Universal Robots URScript: zaboj_fiala_program.script

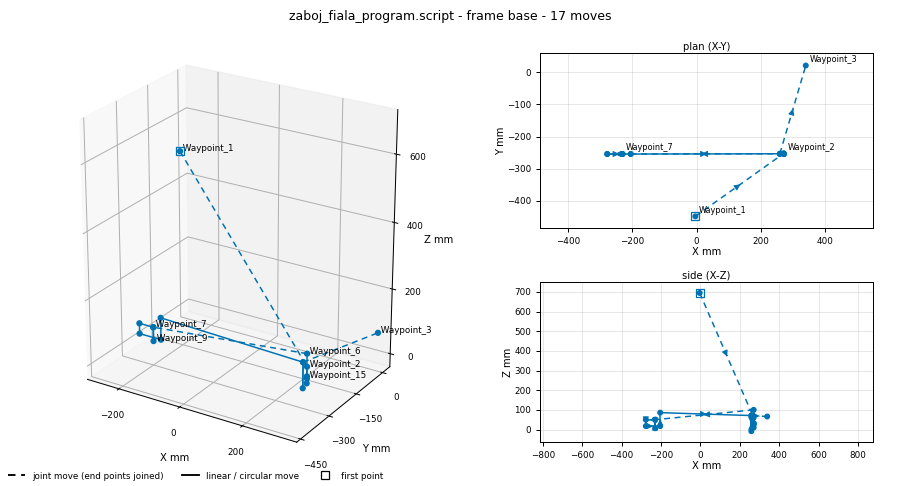
[picture p0: tool path of zaboj_fiala_program.script in frame base, 17 of 20 moves have a stored position in this frame; points joined in program order, loops and branches not executed]
def zaboj_fiala_program():
  global _hidden_verificationVariable=0
  step_count_39f631be_2866_4c45_90c6_6113dbd8747e = 0.0
  thread Step_Counter_Thread_8a2e1a7b_c817_435e_a248_d1a63734bcad():
    while (True):
      step_count_39f631be_2866_4c45_90c6_6113dbd8747e = step_count_39f631be_2866_4c45_90c6_6113dbd8747e + 1.0
      sync()
    end
  end
  run Step_Counter_Thread_8a2e1a7b_c817_435e_a248_d1a63734bcad()
  set_target_payload(1.110000, [0.000000, 0.000000, 0.054000], [0.001832, 0.001832, 0.001832, 0.000000, 0.000000, 0.000000])
  set_gravity([0.0, 0.0, 9.82])
  set_standard_analog_input_domain(0, 1)
  set_standard_analog_input_domain(1, 1)
  set_tool_analog_input_domain(0, 1)
  set_tool_analog_input_domain(1, 1)
  set_analog_outputdomain(0, 1)
  set_analog_outputdomain(1, 1)
  set_input_actions_to_default()
  set_tcp(p[3.414983750301692E-4,-7.378046129560278E-4,0.2251682051354249,-4.265841666109978E-5,-8.612665027929194E-6,-0.002773258026401147])
  set_tool_communication(True, 115200, 0, 1, 1.5, 3.5)
  set_tool_output_mode(0)
  set_tool_digital_output_mode(0, 1)
  set_tool_digital_output_mode(1, 1)
  set_tool_voltage(24)
  set_safety_mode_transition_hardness(1)
  global pocitadlo=7
  global var_2=0
  global referencePoint=p[0.27281535341285135,-0.001324543859192466,-0.05217449401005958,0.008705000024492312,-3.1415499774920335,4.921908573912826E-5]
  global separatorPoint=p[0.0,0.0,0.0,0.0,0.0,0.0]
  # begin: URCap Installation Node
  #   Source: UR Connect, 1.13.79, Universal Robots
  #   Type: UR Connect
  myurRPC = rpc_factory("xmlrpc","http://127.0.0.1:40474")
  # end: URCap Installation Node
  # begin: URCap Installation Node
  #   Source: Robotiq_Grippers, 3.19.1.111718, Robotiq Inc.
  #   Type: Vacuum
  #################################################
  # Vacuum Grip Check
  #################################################

  vacuumGripCheckThread1 = 0
  vacuumGripCheckThread2 = 0
  vacuumGripCheckThread3 = 0
  vacuumGripCheckThread4 = 0
  vacuumGripCheckThread1Running = False
  vacuumGripCheckThread2Running = False
  vacuumGripCheckThread3Running = False
  vacuumGripCheckThread4Running = False
  vacuumGripCheckslave_id = 1
  vacuumGripCheckThreadStarted = False

  thread vacuumGripCheck():
    slave_id = vacuumGripCheckslave_id
    vacuumGripCheckThreadStarted = True

    while (True):
      objectDetectedDebounceCtr = 0

      while (objectDetectedDebounceCtr < 3):
        if(rq_is_vacuum_obj_detected_by_slave_id(slave_id=9)):
          objectDetectedDebounceCtr = objectDetectedDebounceCtr + 1
        else:
          objectDetectedDebounceCtr = 0
        end
        sleep(0.1)
      end

      objectNotDetectedDebounceCtr = 0

      while objectNotDetectedDebounceCtr < 3:
        if (not rq_is_vacuum_obj_detected_by_slave_id(slave_id=9)):
          objectNotDetectedDebounceCtr = objectNotDetectedDebounceCtr + 1
        else:
          objectNotDetectedDebounceCtr = 0
        end
        sleep(0.1)
      end

      socket_open("127.0.0.1",29999,"dashboardServerSocket")
      socket_send_line("pause","dashboardServerSocket")
      socket_send_string("popup Vacuum grip check has detected an object drop.", "dashboardServerSocket")
      socket_send_byte(10, "dashboardServerSocket")
      socket_close("dashboardServerSocket")

      sleep(0.008)
    end
  end

  def startVacuumGripCheckThread(slave_id=9):
    vacuumGripCheckslave_id = slave_id
    threadHandle = run vacuumGripCheck()
    waitForVacuumGripCheckThreadStarted()
    return threadHandle
  end

  def stopVacuumGripCheckThread(threadHandle):
    kill threadHandle
  end

  def waitForVacuumGripCheckThreadStarted():
    while (not(vacuumGripCheckThreadStarted)):
      sleep(0.008)
    end
    vacuumGripCheckThreadStarted = False
  end
  #################################################
  # End - Vacuum Grip Check
  #################################################

  #################################################
  # Stops the pump on a distance travelled
  #################################################
  global stopPumpDistance = 100
  global stopPumpslave_id = 0
  global stopPumpThreadStarted = [False, False, False, False]
  global stopPumpThreadHandles = [0, 0, 0, 0]

  thread stopPumpOnDistanceTravelled():
    distance = stopPumpDistance
    slave_id = stopPumpslave_id
    stopPumpThreadStarted[rq_slave_id_to_index(slave_id)] = True

    measuredDistance = waitForDistanceTravelled(distance)

    rq_stop(slave_id_to_gripper_socket(slave_id))

    stopPumpThreadStarted[rq_slave_id_to_index(slave_id)] = False
  end

  def waitForDistanceTravelled(distance):
    startingPose = get_actual_tcp_pose()
    measuredDistance = 0
    while (measuredDistance < distance):
      sleep(0.1)
      measuredDistance = point_dist(get_actual_tcp_pose(), startingPose)
    end

    return measuredDistance
  end

  def startStopPumpOnDistanceTravelledThread(distance, slave_id=9):
    if (stopPumpThreadStarted[rq_slave_id_to_index(slave_id)]):
      return 0
    end

    global stopPumpDistance = distance
    global stopPumpslave_id = slave_id
    stopPumpThreadHandles[rq_slave_id_to_index(slave_id)] = run stopPumpOnDistanceTravelled()
    waitForStopPumpOnDistanceTravelledThreadStarted(slave_id)
    return stopPumpThreadHandles[rq_slave_id_to_index(slave_id)]
  end

  def waitForStopPumpOnDistanceTravelledThreadStarted(slave_id=9):
    while (not(stopPumpThreadStarted[rq_slave_id_to_index(slave_id)])):
      sleep(0.008)
    end
  end

  def stopStopPumpOnDistanceTravelledThread(slave_id=9):
    handle = stopPumpThreadHandles[rq_slave_id_to_index(slave_id)]
    threadIsRunning = stopPumpThreadStarted[rq_slave_id_to_index(slave_id)]
    if (threadIsRunning):
      kill handle
      stopPumpThreadHandles[rq_slave_id_to_index(slave_id)] = 0
    end
  end
  #################################################
  # End - Stops the pump on a distance travelled
  #################################################

  #################################################
  # Vacuum general functions
  #################################################
  def rq_wait_for_vacuum_object_detected(slave_id=9):
      while (not rq_is_vacuum_obj_detected_by_slave_id(slave_id)):
          if (rq_is_vacuum_timeout(slave_id)):
              return False
          end
          sleep(0.008)
      end
      return True
  end

  def rq_wait_for_vacuum_object_secured(slave_id=9):
      while (not rq_is_vacuum_obj_secured(slave_id)):
          if (rq_is_vacuum_timeout(slave_id)):
              return False
          end
          sleep(0.008)
      end
      return True
  end

  def rq_wait_for_vacuum_object_suction_complete(slave_id=9):
      remaining_retries = 50

       # Wait for suction started
      while (not rq_is_vacuum_obj_in_suction(slave_id) and
             not rq_is_vacuum_obj_detected_by_slave_id(slave_id) and
             remaining_retries > 0):
          sleep(0.01)
          remaining_retries = remaining_retries - 1
      end

      # Wait for suction completed
      while (rq_is_vacuum_obj_in_suction(slave_id)):
          if (rq_is_vacuum_timeout(slave_id)):
              return False
          end
          sleep(0.01)
      end

      return True
  end

  def rq_wait_for_vacuum_object_not_detected(slave_id=9):
      while (rq_is_vacuum_obj_detected_by_slave_id(slave_id)):
          sleep(0.01)
      end
  end

  def rq_is_vacuum_obj_detected_by_slave_id(slave_id=9):
      gOBJ = driver_gripper_client.getObjectDetectionFlag(slave_id)
      return is_vacuum_OBJ_object_detected(gOBJ)
  end

  def rq_is_vacuum_obj_detected(gripper_socket="1"):
      slave_id = gripper_socket_to_slave_id(gripper_socket)
      return rq_is_vacuum_obj_detected_by_slave_id(slave_id)
  end

  def rq_is_vacuum_obj_secured(slave_id=9):
      gOBJ = driver_gripper_client.getObjectDetectionFlag(slave_id)
      return is_vacuum_OBJ_object_secured(gOBJ)
  end

  def rq_is_vacuum_obj_in_suction(slave_id=9):
      gOBJ = driver_gripper_client.getObjectDetectionFlag(slave_id)
      return is_vacuum_OBJ_object_in_motion(gOBJ)
  end

  def rq_is_vacuum_timeout(slave_id=9):
      gFLT = driver_gripper_client.getFault(slave_id)
      return gFLT == 6
  end

  def is_vacuum_OBJ_object_in_motion(gOBJ):
      return gOBJ == 0
  end

  def is_vacuum_OBJ_object_detected(gOBJ):
      return gOBJ == 1 or gOBJ == 2
  end

  def is_vacuum_OBJ_object_secured(gOBJ):
      return gOBJ == 2
  end

  def rq_set_vacuum_and_wait(pressure, timeout, minimum, advanced_mode, slave_id=9):
      driver_gripper_client.configureVacuum(slave_id, advanced_mode, pressure, minimum, timeout)
  end

  def is_continuous_grip(maximum_vacuum):
    return maximum_vacuum == 0
  end

  def rq_vacuum_release(advanced_mode=False, shutoff_distance_cm=5, wait_for_object_released=True, gripper_socket="1"):
    rq_wait_for_gripper_reconnection()
    local slave_id = gripper_socket_to_slave_id(gripper_socket)
    local shutoff_distance = scale(shutoff_distance_cm, [0, 99], [0.00, 0.99])
    local pressure = 255
    local minimum = 0
    local timeout = 255
    rq_vacuum_release_raw(advanced_mode, pressure, minimum, timeout, shutoff_distance, wait_for_object_released, slave_id)
  end

  def rq_vacuum_release_raw(advanced_mode, pressure, minimum, timeout, shutoff_distance, wait_for_object_released, slave_id):
    rq_reset_fault_and_activate(slave_id)

    if advanced_mode:
      rq_set_vacuum_and_wait(pressure, timeout, minimum, 1, slave_id)
    else:
      rq_set_vacuum_and_wait(pressure, timeout, minimum, 0, slave_id)
    end

    # The following patch is for Robotiq's Camera issue when communication is lost, but not the activation
    # the communication driver reset the GTO bit
    driver_gripper_client.goto(slave_id, 1)

    if wait_for_object_released:
      while (rq_is_vacuum_obj_detected_by_slave_id(slave_id)):

        if advanced_mode:
          rq_set_vacuum_and_wait(pressure, timeout, minimum, 1, slave_id)
        else:
          rq_set_vacuum_and_wait(pressure, timeout, minimum, 0, slave_id)
        end

        # The following patch is for Robotiq's Camera issue when communication is lost, but not the activation
        # the communication driver reset the GTO bit
        driver_gripper_client.goto(slave_id, 1)
        sleep(0.01)
      end
    end

    if advanced_mode:
      startStopPumpOnDistanceTravelledThread(shutoff_distance, slave_id)
    end
  end

  def rq_vacuum_grip(advanced_mode=False, maximum_vacuum=60, minimum_vacuum=40, timeout_ms=3000, wait_for_object_detected=True, gripper_socket="1"):
    rq_wait_for_gripper_reconnection()
    local slave_id = gripper_socket_to_slave_id(gripper_socket)
    local pressure = floor(scale(maximum_vacuum, [0, 100], [100, 0]))
    local minimum = floor(scale(minimum_vacuum, [0, 100], [100, 0]))
    local timeout = floor(scale(timeout_ms, [0, 25500], [0, 255]))
    rq_vacuum_grip_raw(advanced_mode, pressure, minimum, timeout, slave_id)
    if wait_for_object_detected:
          suction_completed = rq_wait_for_vacuum_object_suction_complete(slave_id)
          if(not suction_completed):
            driver_gripper_client.goto(slave_id, 0)
          end
    end
  end

  def rq_vacuum_grip_raw(advanced_mode, pressure, minimum, timeout, slave_id):
    stopStopPumpOnDistanceTravelledThread(slave_id)
    rq_reset_fault_and_activate(slave_id)

    if advanced_mode:
      rq_set_vacuum_and_wait(pressure, timeout, minimum, 1, slave_id)
    else:
      rq_set_vacuum_and_wait(pressure, timeout, minimum, 0, slave_id)
    end

    driver_gripper_client.goto(slave_id, 1)
  end

  def is_FLT_no_fault(gFLT):
      return gFLT == 0
  end

  def is_FLT_vacuum_timeout(gFLT):
    return gFLT == 6
  end

  def is_FLT_faulted(gFLT):
      return gFLT >= 8
  end

  def rq_reset_fault_and_activate(slave_id):
      gFLT = driver_gripper_client.getFault(slave_id)

      if(not is_FLT_no_fault(gFLT)):
          if(is_FLT_vacuum_timeout(gFLT)):
              driver_gripper_client.goto(slave_id, 0)
          elif(is_FLT_faulted(gFLT)):
              driver_gripper_client.goto(slave_id, 0)
              driver_gripper_client.activate([slave_id], True)
          end
      elif(not rq_is_gripper_activated(slave_id)):
          driver_gripper_client.goto(slave_id, 0)
          driver_gripper_client.activate([slave_id], False)
      end
  end
  #################################################
  # End - Vacuum general functions
  #################################################
    def scale(value, rawRange, scaledRange):
        def computeSlope(inputRange, outputRange):
            outputRangeDelta = outputRange[1] - outputRange[0]
            inputRangeDelta = inputRange[1] - inputRange[0]

            if (inputRangeDelta == 0):
                return 0
            else:
                return outputRangeDelta / inputRangeDelta
            end
        end

        def computeIntercept(slope, inputRange, outputRange):
            return outputRange[0] - (slope * inputRange[0])
        end

        def clipScaledValue(outputScaledValue, outputRange):
            if (outputRange[0] < outputRange[1]):
                return clipWhenLowerLimitIsLessThanHigher(outputScaledValue, outputRange)
            else:
                return clipWhenLowerLimitIsGreaterThanHigherLimit(outputScaledValue, outputRange)
            end
        end

        def clipWhenLowerLimitIsGreaterThanHigherLimit(outputScaledValue, outputRange):
            if (outputScaledValue < outputRange[1]):
                return outputRange[1]
            elif (outputScaledValue > outputRange[0]):
                return outputRange[0]
            else:
                return outputScaledValue
            end
        end

        def clipWhenLowerLimitIsLessThanHigher(outputScaledValue, outputRange):
            if (outputScaledValue < outputRange[0]):
                return outputRange[0]
            elif (outputScaledValue > outputRange[1]):
                return outputRange[1]
            else:
                return outputScaledValue
            end
        end

        slope = computeSlope(rawRange, scaledRange)
        intercept = computeIntercept(slope, rawRange, scaledRange)
        scaledValue = slope * value + intercept
        return clipScaledValue(scaledValue, scaledRange)
    end

    def limit(value, range):
        return scale(value, range, range)
    end

  vacuumGripCheckWarningTitle = "Vacuum grip check"
  vacuumGripCheckWarningMessage = "Vacuum gripper object lost"
  vacuumGripTimeoutTitle = "Vacuum gripper fault"
  vacuumGripTimeoutMessage = "Grip has timed out"
  # end: URCap Installation Node
  # begin: URCap Installation Node
  #   Source: Robotiq_Grippers, 3.19.1.111718, Robotiq Inc.
  #   Type: Gripper
  RQ_UNIT_PERCENT = 0
  RQ_UNIT_MM = 1
  RQ_UNIT_INCH = 2

  global gripper_reconnecting = False
  rq_current_limit_enabled = False
  gripper_closed_norm = [100, 100, 100, 100]
  gripper_open_norm = [0, 0, 0, 0]
  gripper_closed_mm = [0, 0, 0, 0]
  gripper_open_mm = [50, 50, 50, 50]

  driver_gripper_client = rpc_factory("xmlrpc","http://127.0.0.1:63353")

  def rq_set_force_norm(force_norm, gripper_socket="1"):
      rq_wait_for_gripper_reconnection()
      slave_id = gripper_socket_to_slave_id(gripper_socket)
      rq_set_force_norm_multi_grippers(force_norm, [slave_id])
  end

  def rq_set_force_norm_multi_grippers(force_norm, slave_ids=[9]):
      driver_gripper_client.setForce(slave_ids, force_norm)
  end

  def rq_set_speed_norm(speed_norm, gripper_socket="1"):
      rq_wait_for_gripper_reconnection()
      slave_id = gripper_socket_to_slave_id(gripper_socket)
      rq_set_speed_norm_multi_grippers(speed_norm, [slave_id])
  end

  def rq_set_speed_norm_multi_grippers(speed_norm, slave_ids=[9]):
      driver_gripper_client.setSpeed(slave_ids, speed_norm)
  end

  def rq_open_and_wait(gripper_socket="1"):
      rq_wait_for_gripper_reconnection()
      slave_id = gripper_socket_to_slave_id(gripper_socket)
      driver_gripper_client.openGripper(slave_id)
      rq_wait_for_motion_complete([slave_id])
  end

  def rq_close_and_wait(gripper_socket="1"):
      rq_wait_for_gripper_reconnection()
      slave_id = gripper_socket_to_slave_id(gripper_socket)
      driver_gripper_client.closeGripper(slave_id)
      rq_wait_for_motion_complete([slave_id])
  end

  def rq_move_norm_multi_grippers(position, slave_ids=[9]):
     # rq_wait_for_gripper_reconnection fucntion is not called here because it is already done in the gripper contribution
     # script and this function is not defined for public usage.
     all_gripper_limits = get_all_gripper_limits(slave_ids)
     driver_gripper_client.move(slave_ids, position, RQ_UNIT_PERCENT, all_gripper_limits)
  end

  def rq_move_and_wait_norm_multi_grippers(position, slave_ids=[9]):
       all_gripper_limits = get_all_gripper_limits(slave_ids)
       driver_gripper_client.move(slave_ids, position, RQ_UNIT_PERCENT, all_gripper_limits)
       rq_wait_for_motion_complete(slave_ids)
  end

  def rq_move_and_wait(position, unit, gripper_socket="1"):
     rq_wait_for_gripper_reconnection()
     slave_id = gripper_socket_to_slave_id(to_str(gripper_socket))
     all_gripper_limits = get_all_gripper_limits([slave_id])
     driver_gripper_client.move([slave_id], position, unit, all_gripper_limits)
     rq_wait_for_motion_complete([slave_id])
  end

  def rq_move_and_wait_norm(position, gripper_socket="1"):
      rq_move_and_wait(position, RQ_UNIT_PERCENT, gripper_socket)
  end

  def rq_move_and_wait_mm(position, gripper_socket="1"):
      rq_move_and_wait(position, RQ_UNIT_MM, gripper_socket)
  end

  def rq_move_and_wait_inches(position, gripper_socket="1"):
     rq_move_and_wait(position, RQ_UNIT_INCH, gripper_socket)
  end

  def rq_is_object_detected(gripper_socket="1"):
     slave_id = gripper_socket_to_slave_id(gripper_socket)
     return driver_gripper_client.isObjectDetected(slave_id)
  end

  def rq_current_pos_norm(gripper_socket="1"):
      slave_id = gripper_socket_to_slave_id(gripper_socket)
      gripper_limits = get_gripper_limits(gripper_socket)
      return driver_gripper_client.getCurrentPosition(slave_id,
                                    RQ_UNIT_PERCENT,
                                    gripper_limits[0],
                                    gripper_limits[1],
                                    gripper_limits[2],
                                    gripper_limits[3])
  end

  def rq_current_pos_mm(gripper_socket=1):
      slave_id = gripper_socket_to_slave_id(to_str(gripper_socket))
      gripper_limits = get_gripper_limits(to_str(gripper_socket))
      return driver_gripper_client.getCurrentPosition(slave_id,
                                    RQ_UNIT_MM,
                                    gripper_limits[0],
                                    gripper_limits[1],
                                    gripper_limits[2],
                                    gripper_limits[3])
  end

  def rq_current_pos_inches(gripper_socket=1):
      slave_id = gripper_socket_to_slave_id(to_str(gripper_socket))
      gripper_limits = get_gripper_limits(to_str(gripper_socket))
      return driver_gripper_client.getCurrentPosition(slave_id,
                                    RQ_UNIT_INCH,
                                    gripper_limits[0],
                                    gripper_limits[1],
                                    gripper_limits[2],
                                    gripper_limits[3])
  end

  def rq_reset(gripper_socket="1"):
      slave_id = gripper_socket_to_slave_id(gripper_socket)
      driver_gripper_client.deactivate([slave_id])
  end

  def rq_set_gripper_max_cur(current_mA, gripper_socket="1"):
      rq_wait_for_gripper_reconnection()
      slave_id = gripper_socket_to_slave_id(gripper_socket)
      driver_gripper_client.setMaximumCurrent(current_mA, slave_id)
  end

  def rq_get_gripper_max_cur(gripper_socket="1"):
      slave_id = gripper_socket_to_slave_id(gripper_socket)
      return driver_gripper_client.getMaximumCurrent(slave_id)
  end

  def rq_set_max_current_for_all_grippers():
      rq_wait_for_gripper_reconnection()
      driver_gripper_client.setMaximumCurrentOnAllGrippers(rq_current_limit_enabled)
  end

  def rq_is_gripper_activated(slave_id=9):
      return driver_gripper_client.isGripperActivated(slave_id)
  end

  def rq_is_gripper_connected(slave_id=9):
      return driver_gripper_client.isGripperConnected(slave_id)
  end

  def rq_get_fault(slave_id=9):
      return driver_gripper_client.getFault(slave_id)
  end

  def rq_activate_and_wait(gripper_socket="1"):
      slave_id = gripper_socket_to_slave_id(gripper_socket)
      if (not rq_is_gripper_activated(slave_id)):
        driver_gripper_client.activate([slave_id], False)
      end
  end

  def rq_activate_all_grippers(reset=False):
      empty_array_used_to_act_on_all_grippers = []
      if (reset):
        driver_gripper_client.activate(empty_array_used_to_act_on_all_grippers, True)
      else:
        driver_gripper_client.activateIfRequired(empty_array_used_to_act_on_all_grippers)
      end
  end

  def get_closed_norm(gripper_socket):
      return gripper_closed_norm[rq_gripper_socket_to_index(gripper_socket)]
  end

  def get_open_norm(gripper_socket):
      return gripper_open_norm[rq_gripper_socket_to_index(gripper_socket)]
  end

  def get_open_mm(gripper_socket):
      return gripper_open_mm[rq_gripper_socket_to_index(gripper_socket)]
  end

  def get_closed_mm(gripper_socket):
      return gripper_closed_mm[rq_gripper_socket_to_index(gripper_socket)]
  end

  def set_closed_norm(closed_norm, gripper_socket):
      gripper_closed_norm[rq_gripper_socket_to_index(gripper_socket)] = closed_norm
  end

  def set_open_norm(open_norm, gripper_socket):
      gripper_open_norm[rq_gripper_socket_to_index(gripper_socket)] = open_norm
  end

  def set_closed_mm(closed_mm, gripper_socket):
      gripper_closed_mm[rq_gripper_socket_to_index(gripper_socket)] = closed_mm
  end

  def set_open_mm(opened_mm, gripper_socket):
      gripper_open_mm[rq_gripper_socket_to_index(gripper_socket)] = opened_mm
  end

  def slave_id_to_gripper_socket(slave_id):
      if slave_id == 9:
          return "1"
      else:
          return to_str(slave_id)
      end
  end

  def gripper_socket_to_slave_id(gripper_socket):
      if gripper_socket == "1":
          return 9
      else:
          return to_num(gripper_socket)
      end
  end

  def rq_slave_id_to_index(slave_id):
      if slave_id == 9:
          return 0
      else:
          return slave_id - 1
      end
  end

  def rq_gripper_socket_to_index(gripper_socket):
      return to_num(gripper_socket) - 1
  end

  def get_all_gripper_limits(slave_ids):
     all_gripper_limits = [0, 0, 0, 0, 0, 0, 0, 0, 0, 0, 0, 0, 0, 0, 0, 0]
     nb_slave_ids = get_list_length(slave_ids)
     slave_id_index = 0
     index = 0
     sub_index = 0
     while (index < nb_slave_ids):
         slave_id_index = 0
         items_per_limit = 4
         gripper_socket = slave_id_to_gripper_socket(slave_ids[index])
         gripper_limits = get_gripper_limits(gripper_socket)
         while (sub_index < items_per_limit):
            all_gripper_limits[index] = gripper_limits[sub_index]
            sub_index = sub_index + 1
            index = index + 1
         end
         index = index + 1
     end

     return all_gripper_limits
  end

  def get_gripper_limits(gripper_socket):
      return [get_closed_norm(gripper_socket),
              get_open_norm(gripper_socket),
              get_closed_mm(gripper_socket),
              get_open_mm(gripper_socket)]
  end

  def rq_wait_for_motion_complete(slave_ids):
      nb_slave_ids = get_list_length(slave_ids)
      index = 0
      while (index < nb_slave_ids):
        rq_wait(slave_ids[index])
        index = index + 1
      end
  end

  def rq_stop(gripper_socket="1"):
      slave_id = gripper_socket_to_slave_id(gripper_socket)
      driver_gripper_client.goto(slave_id, 0)
  end

  def rq_wait(slave_id):
      # Wait for the gripper motion to complete
      while (not rq_is_motion_complete(slave_id)):
          # The following patch is for Robotiq's Camera issue when communication is lost, but not the activation
          # the communication driver reset the GTO bit
          driver_gripper_client.goto(slave_id, 1)
          sleep(0.1)
      end
  end

  def rq_is_motion_complete(slave_id):
      detection_flag = driver_gripper_client.getObjectDetectionFlag(slave_id)
      return detection_flag > 0 and detection_flag < 4
  end

  def write_error_popup(index, message_part_1, message_part_2, title):
      popup_message_part_1 = str_cat(message_part_1, index)
      popup_message_part_2 = str_cat(popup_message_part_1, " ")
      popup_message = str_cat(popup_message_part_2, message_part_2)
      return popup(popup_message, title, False, True, True)
  end

  def rq_disconnect_grippers():
      driver_gripper_client.pauseAndDisconnect()
  end

  def rq_reconnect_grippers(blocking=False, slave_ids=[]):
      if blocking:
          global gripper_reconnecting = True
          driver_gripper_client.reconnectAndResume(slave_ids)
          gripper_reconnecting = False
      else:
          thread recon_thread():
              rq_reconnect_grippers(True)
              return False
          end
          thrd = run recon_thread()
      end
  end

  def rq_wait_for_gripper_reconnection(timeout_s = 30.0):
      while (gripper_reconnecting == True):
          if (timeout_s <= 0):
            popup("Gripper has not reconnected before the expected time")
            halt
          else:
            sync()
            timeout_s = timeout_s - get_steptime()
          end
      end
  end

  def rq_gripper_allow_tool_com(allow_tool_comm):
      driver_gripper_client.allowToolComm(allow_tool_comm)
  end
  set_closed_norm(100.0, "1")
  set_open_norm(0.0, "1")
  set_closed_mm(0.0, "1")
  set_open_mm(50.0, "1")
  set_closed_norm(100.0, "2")
  set_open_norm(0.0, "2")
  set_closed_mm(0.0, "2")
  set_open_mm(50.0, "2")
  set_closed_norm(100.0, "3")
  set_open_norm(0.0, "3")
  set_closed_mm(0.0, "3")
  set_open_mm(50.0, "3")
  set_closed_norm(100.0, "4")
  set_open_norm(0.0, "4")
  set_closed_mm(0.0, "4")
  set_open_mm(50.0, "4")
  rq_current_limit_enabled = False
  # end: URCap Installation Node
  global Pallet_1_cnt=1
  global Pallet_1_lct=1
  global Pallet_1_lno=1
  global Pallet_1_sep= False
  global Pallet_1_tct=1
  global qNearApproach=[0,0,0,0,0,0]
  global Waypoint_1_p=p[-.003732499146, -.447764350544, .694668676500, .010357527271, 2.217455435209, -2.215428702531]
  global Waypoint_1_q=[0.004420539364218712, -1.5699242066223924, 0.010914627705709279, -1.5611537259868165, -0.009149853383199513, -0.008998696004049123]
  global Waypoint_2_p=p[.270561572388, -.252460408212, .060750519249, -2.205633529341, 2.237137668558, .000000000220]
  global Waypoint_2_q=[-0.38798117147393185, -1.7670171967297028, -1.4314454771594134, -1.5127431085216578, 1.5630238713731401, -0.37426215443183697]
  global Waypoint_15_p=p[.270561572385, -.252460408216, .025108204613, -2.205633532066, 2.237137671479, .000000000266]
  global Waypoint_15_q=[-0.387640232785321, -1.7878663927529868, -1.574689349085693, -1.3486454019375724, 1.5632032959842548, -0.37526689414023995]
  global Waypoint_4_p=p[.271723132448, -.254713739484, .032576839225, -2.202352738203, 2.233984750329, -.017109190704]
  global Waypoint_4_q=[-0.39231975839608957, -1.777546052304718, -1.5566950178122445, -1.365160337822867, 1.5630833526801635, -0.37973253437504706]
  global Waypoint_5_p=p[.270561572159, -.253261773950, .010467803518, -2.205633542175, 2.237137697756, .000000006507]
  global Waypoint_5_q=[-0.3896634195662285, -1.805539464463246, -1.6233792723820244, -1.2822808384995135, 1.5633685440948906, -0.377819460409726]
  global Waypoint_6_p=p[.270561572150, -.253261773946, .100610117048, -2.205633531713, 2.237137687145, .000000006506]
  global Waypoint_6_q=[-0.39059338186191184, -1.7752166803415488, -1.2341938193302262, -1.7018008441992443, 1.5631981308940244, -0.3753075181511152]
  global Waypoint_7_p=p[-.230058808373, -.254188582133, .050546411075, -2.205633551354, 2.237137688707, -.000000002111]
  global Waypoint_7_q=[-1.9158549360473138, -1.6556048584721488, -1.6085609835301513, -1.4470858589855453, 1.5627141197324992, -1.9027213849297713]
  global Waypoint_9_p=p[-.230058808390, -.254188582182, .007047120969, -2.205633540891, 2.237137678096, -.000000002113]
  global Waypoint_9_q=[-1.9154641598153326, -1.6964409636789144, -1.7725358360043462, -1.2422691400022003, 1.563132548677892, -1.9039956648963363]
  global Waypoint_11_p=p[-.277401121907, -.254188582125, .050546411070, -2.205633551354, 2.237137688707, -.000000002111]
  global Waypoint_11_q=[-2.045659040969955, -1.8025670740351707, -1.4352832270086573, -1.4734087088425873, 1.5631794833456076, -2.0322455626523688]
  global Waypoint_12_p=p[-.277401121893, -.254188582096, .018070817914, -2.205633540892, 2.237137678095, -.000000002109]
  global Waypoint_12_q=[-2.045358845597888, -1.825729367137832, -1.5604181602870781, -1.3251075677590576, 1.5633936278058413, -2.0331527047927835]
  global Waypoint_13_p=p[-.204474181310, -.254188582073, .018070817902, -2.205633551354, 2.237137688706, -.000000002109]
  global Waypoint_13_q=[-1.8362919914072373, -1.6095973638389953, -1.8134970852229308, -1.288148318123807, 1.5627547664611345, -1.8244687075886024]
  global Waypoint_14_p=p[-.204474181308, -.254188582064, .086413131433, -2.205633551354, 2.237137688706, -.000000002108]
  global Waypoint_14_q=[-1.8369625886427805, -1.574832125077247, -1.5248047019871604, -1.6116166051216325, 1.5624717189936659, -1.8224669010736845]
  global Waypoint_8_p=p[.258569396158, -.253443601432, .071606282054, -2.202406735368, 2.240314480847, -.000000000314]
  global Waypoint_8_q=[-0.4042975507105382, -1.7298519365980187, -1.4251167858707436, -1.5562383352509102, 1.5629115038954633, -0.38735228726952897]
  global Waypoint_10_p=p[.258569396172, -.253443601435, -.007836031423, -2.202406734996, 2.240314481213, -.000000000000]
  global Waypoint_10_q=[-0.4035716267056175, -1.7950209472926995, -1.7277873303001208, -1.1883889938254129, 1.5635490193420658, -0.3896017747848468]
  global Waypoint_3_p=p[.339173069408, .020646450111, .066698974081, -.046899901835, 3.140174557594, -.015225451020]
  global Waypoint_3_q=[0.46848809719085693, -1.6360541782774867, -1.5524871349334717, -1.5260256093791504, 1.5533761978149414, 2.0090246200561523]
  global Approach_p=p[.272815353377, -.001324543879, -.033905691191, .008705000027, -3.141549977485, .000049219079]
  global Approach_q=[0.5000229007972248, -1.457555270442966, -2.2252279375503816, -1.0285170994385489, 1.5629147840442803, 2.0609351731087564]
  global ToolActionPoint_p=p[.272815353413, -.001324543859, -.052174494010, .008705000022, -3.141549977485, .000049219087]
  global ToolActionPoint_q=[0.500250470542329, -1.5124229690085453, -2.280892902919593, -0.9179415944854314, 1.5635788131215058, 2.060298978026008]
  global Exit_1_p=p[.272815353404, -.001324543864, .045467820739, .008705000021, -3.141549977496, .000049219082]
  global Exit_1_q=[0.49925098394912215, -1.3352160082302609, -1.9246151993381408, -1.4514821535151832, 1.5615809977592896, 2.0636040213119218]
  $ 2 "BeforeStart"
  # begin: URCap Program Node
  #   Source: Robotiq_Grippers, 3.19.1.111718, Robotiq Inc.
  #   Type: Gripper Activate
  $ 3 "Gripper Reset and Activate"

  rq_set_max_current_for_all_grippers()

  reset_and_activate = True

  rq_activate_all_grippers(True)
  # end: URCap Program Node
  $ 4 "MoveJ"
  $ 5 "Waypoint_1" "breakAfter"
  movej(get_inverse_kin(Waypoint_1_p, qnear=Waypoint_1_q), a=1.3962634015954636, v=1.0471975511965976)
  $ 6 "Wait Sensor_vzadu=HI"
  while (get_standard_digital_in(2) == False):
    sync()
  end
  $ 66 "Thread_1"
  thread Thread_1():
    while (True):
      $ 67 "Set Dopravnik=On"
      set_standard_digital_out(2, True)
      $ 68 "Wait Sensor_vzadu=HI"
      while (get_standard_digital_in(2) == False):
        sync()
      end
      $ 69 "Set Dopravnik=Off"
      set_standard_digital_out(2, False)
      $ 70 "Wait Sensor_vzadu=LO"
      while (get_standard_digital_in(2) == True):
        sync()
      end
      $ 71 "Wait: 1.0"
      sleep(1.0)
    end
  end
  threadId_Thread_1 = run Thread_1()
  while (True):
    $ 7 "Robot Program"
    $ 8 "MoveJ"
    $ 9 "Waypoint_2" "breakAfter"
    movej(get_inverse_kin(Waypoint_2_p, qnear=Waypoint_2_q), a=1.3962634015954636, v=1.0471975511965976)
    $ 10 "Wait Sensor_vzadu=HI"
    while (get_standard_digital_in(2) == False):
      sync()
    end
    # begin: URCap Program Node
    #   Source: Robotiq_Grippers, 3.19.1.111718, Robotiq Inc.
    #   Type: Gripper
    $ 11 "Gripper Close (1)"
    gripper_slave_ids_0 = [9]
    popupErrorGripperWord = "Gripper"
    popupErrorNoConnection1 = "must be connected to run this program."
    popupErrorNoConnection2 = "No connection"
    popupErrorNotActivated1 = "is not activated. Go to Installation tab > Gripper to activate it and run the program again."
    popupErrorNotActivated2 = "Not activated"
    rq_gripper_speed = 100.0
    rq_gripper_force = 20.0
    rq_gripper_position = 100.0
    rq_is_blocking = True
    rq_is_robot_compliant = False
    nb_slave_ids = get_list_length(gripper_slave_ids_0)
    rq_wait_for_gripper_reconnection()
    index = 0
    while (index < nb_slave_ids):
        if (not rq_is_gripper_connected(gripper_slave_ids_0[index])):
            write_error_popup(index, popupErrorGripperWord, popupErrorNoConnection1, popupErrorNoConnection2)
        end
        index = index + 1
    end
    index = 0
    while (index < nb_slave_ids):
        if (not rq_is_gripper_activated(gripper_slave_ids_0[index])):
            write_error_popup(index, popupErrorGripperWord, popupErrorNotActivated1, popupErrorNotActivated2)
        end
        index = index + 1
    end
    rq_set_speed_norm_multi_grippers(rq_gripper_speed, gripper_slave_ids_0)
    rq_set_force_norm_multi_grippers(rq_gripper_force, gripper_slave_ids_0)
    if (rq_is_blocking):
        if rq_is_robot_compliant:
            zero_ftsensor()
            sleep(0.02)
            # Maximum allowed deviation values for non-compliant axes are default values generated by UR in a Force node
            force_mode(tool_pose(), [1, 1, 0, 0, 0, 0], [0.0, 0.0, 0.0, 0.0, 0.0, 0.0], 2, [0.15, 0.15, 0.1, 0.3490658503988659, 0.3490658503988659, 0.3490658503988659])
        end
        rq_move_and_wait_norm_multi_grippers(rq_gripper_position, gripper_slave_ids_0)
        if rq_is_robot_compliant:
            end_force_mode()
        end
    else:
        rq_move_norm_multi_grippers(rq_gripper_position, gripper_slave_ids_0)
    end
    # end: URCap Program Node
    $ 12 "MoveL"
    $ 13 "Waypoint_15" "breakAfter"
    movel(Waypoint_15_p, a=1.2, v=0.05)
    $ 14 "var_1≔force()"
    global var_1= force ()
    $ 15 "MoveL"
    $ 16 "Waypoint_4" "breakAfter"
    movel(Waypoint_4_p, a=1.2, v=0.25)
    $ 17 "If var_1>5"
    if (var_1>5):
      $ 18 "MoveL"
      # begin: URCap Program Node
      #   Source: Robotiq_Grippers, 3.19.1.111718, Robotiq Inc.
      #   Type: Gripper
      $ 19 "Gripper Open (1)"
      gripper_slave_ids_1 = [9]
      popupErrorGripperWord = "Gripper"
      popupErrorNoConnection1 = "must be connected to run this program."
      popupErrorNoConnection2 = "No connection"
      popupErrorNotActivated1 = "is not activated. Go to Installation tab > Gripper to activate it and run the program again."
      popupErrorNotActivated2 = "Not activated"
      rq_gripper_speed = 100.0
      rq_gripper_force = 20.0
      rq_gripper_position = 0.0
      rq_is_blocking = True
      rq_is_robot_compliant = False
      nb_slave_ids = get_list_length(gripper_slave_ids_1)
      rq_wait_for_gripper_reconnection()
      index = 0
      while (index < nb_slave_ids):
          if (not rq_is_gripper_connected(gripper_slave_ids_1[index])):
              write_error_popup(index, popupErrorGripperWord, popupErrorNoConnection1, popupErrorNoConnection2)
          end
          index = index + 1
      end
      index = 0
      while (index < nb_slave_ids):
          if (not rq_is_gripper_activated(gripper_slave_ids_1[index])):
              write_error_popup(index, popupErrorGripperWord, popupErrorNotActivated1, popupErrorNotActivated2)
          end
          index = index + 1
      end
      rq_set_speed_norm_multi_grippers(rq_gripper_speed, gripper_slave_ids_1)
      rq_set_force_norm_multi_grippers(rq_gripper_force, gripper_slave_ids_1)
      if (rq_is_blocking):
          if rq_is_robot_compliant:
              zero_ftsensor()
              sleep(0.02)
              # Maximum allowed deviation values for non-compliant axes are default values generated by UR in a Force node
              force_mode(tool_pose(), [1, 1, 0, 0, 0, 0], [0.0, 0.0, 0.0, 0.0, 0.0, 0.0], 2, [0.15, 0.15, 0.1, 0.3490658503988659, 0.3490658503988659, 0.3490658503988659])
          end
          rq_move_and_wait_norm_multi_grippers(rq_gripper_position, gripper_slave_ids_1)
          if rq_is_robot_compliant:
              end_force_mode()
          end
      else:
          rq_move_norm_multi_grippers(rq_gripper_position, gripper_slave_ids_1)
      end
      # end: URCap Program Node
      $ 20 "Waypoint_5" "breakAfter"
      movel(Waypoint_5_p, a=1.2, v=0.25)
      # begin: URCap Program Node
      #   Source: Robotiq_Grippers, 3.19.1.111718, Robotiq Inc.
      #   Type: Gripper
      $ 21 "Gripper Close (1)"
      gripper_slave_ids_2 = [9]
      popupErrorGripperWord = "Gripper"
      popupErrorNoConnection1 = "must be connected to run this program."
      popupErrorNoConnection2 = "No connection"
      popupErrorNotActivated1 = "is not activated. Go to Installation tab > Gripper to activate it and run the program again."
      popupErrorNotActivated2 = "Not activated"
      rq_gripper_speed = 100.0
      rq_gripper_force = 20.0
      rq_gripper_position = 100.0
      rq_is_blocking = True
      rq_is_robot_compliant = False
      nb_slave_ids = get_list_length(gripper_slave_ids_2)
      rq_wait_for_gripper_reconnection()
      index = 0
      while (index < nb_slave_ids):
          if (not rq_is_gripper_connected(gripper_slave_ids_2[index])):
              write_error_popup(index, popupErrorGripperWord, popupErrorNoConnection1, popupErrorNoConnection2)
          end
          index = index + 1
      end
      index = 0
      while (index < nb_slave_ids):
          if (not rq_is_gripper_activated(gripper_slave_ids_2[index])):
              write_error_popup(index, popupErrorGripperWord, popupErrorNotActivated1, popupErrorNotActivated2)
          end
          index = index + 1
      end
      rq_set_speed_norm_multi_grippers(rq_gripper_speed, gripper_slave_ids_2)
      rq_set_force_norm_multi_grippers(rq_gripper_force, gripper_slave_ids_2)
      if (rq_is_blocking):
          if rq_is_robot_compliant:
              zero_ftsensor()
              sleep(0.02)
              # Maximum allowed deviation values for non-compliant axes are default values generated by UR in a Force node
              force_mode(tool_pose(), [1, 1, 0, 0, 0, 0], [0.0, 0.0, 0.0, 0.0, 0.0, 0.0], 2, [0.15, 0.15, 0.1, 0.3490658503988659, 0.3490658503988659, 0.3490658503988659])
          end
          rq_move_and_wait_norm_multi_grippers(rq_gripper_position, gripper_slave_ids_2)
          if rq_is_robot_compliant:
              end_force_mode()
          end
      else:
          rq_move_norm_multi_grippers(rq_gripper_position, gripper_slave_ids_2)
      end
      # end: URCap Program Node
      $ 22 "SetPayloadNode: {PayloadReferenceComponent; InstallationPayloadComponent name=Payload_brick; contributorInfo=com.ur.polyscope.payload.common.InstallationPayloadComponent$1@50a04d; mass=1.18 kg; centerOfGravity=(0.003, -0.002, 0.05); Ixx=0.002028, Iyy=0.002028, Izz=0.002028, Ixy=0.000000, Ixz=0.000000, Iyz=0.000000, transitionTime: 0.05 s}"
      set_target_payload(1.180000, [0.003000, -0.002000, 0.050000], [0.002028, 0.002028, 0.002028, 0.000000, 0.000000, 0.000000], 0.050000)
      $ 23 "Waypoint_6" "breakAfter"
      movel(Waypoint_6_p, a=1.2, v=0.25)
      $ 24 "MoveJ"
      $ 25 "Waypoint_7" "breakAfter"
      movej(get_inverse_kin(Waypoint_7_p, qnear=Waypoint_7_q), a=1.3962634015954636, v=1.0471975511965976)
      $ 26 "MoveL"
      $ 27 "Waypoint_9" "breakAfter"
      movel(Waypoint_9_p, a=1.2, v=0.25)
      # begin: URCap Program Node
      #   Source: Robotiq_Grippers, 3.19.1.111718, Robotiq Inc.
      #   Type: Gripper
      $ 28 "Gripper Open (1)"
      gripper_slave_ids_3 = [9]
      popupErrorGripperWord = "Gripper"
      popupErrorNoConnection1 = "must be connected to run this program."
      popupErrorNoConnection2 = "No connection"
      popupErrorNotActivated1 = "is not activated. Go to Installation tab > Gripper to activate it and run the program again."
      popupErrorNotActivated2 = "Not activated"
      rq_gripper_speed = 20.0
      rq_gripper_force = 100.0
      rq_gripper_position = 0.0
      rq_is_blocking = True
      rq_is_robot_compliant = False
      nb_slave_ids = get_list_length(gripper_slave_ids_3)
      rq_wait_for_gripper_reconnection()
      index = 0
      while (index < nb_slave_ids):
          if (not rq_is_gripper_connected(gripper_slave_ids_3[index])):
              write_error_popup(index, popupErrorGripperWord, popupErrorNoConnection1, popupErrorNoConnection2)
          end
          index = index + 1
      end
      index = 0
      while (index < nb_slave_ids):
          if (not rq_is_gripper_activated(gripper_slave_ids_3[index])):
              write_error_popup(index, popupErrorGripperWord, popupErrorNotActivated1, popupErrorNotActivated2)
          end
          index = index + 1
      end
      rq_set_speed_norm_multi_grippers(rq_gripper_speed, gripper_slave_ids_3)
      rq_set_force_norm_multi_grippers(rq_gripper_force, gripper_slave_ids_3)
      if (rq_is_blocking):
          if rq_is_robot_compliant:
              zero_ftsensor()
              sleep(0.02)
              # Maximum allowed deviation values for non-compliant axes are default values generated by UR in a Force node
              force_mode(tool_pose(), [1, 1, 0, 0, 0, 0], [0.0, 0.0, 0.0, 0.0, 0.0, 0.0], 2, [0.15, 0.15, 0.1, 0.3490658503988659, 0.3490658503988659, 0.3490658503988659])
          end
          rq_move_and_wait_norm_multi_grippers(rq_gripper_position, gripper_slave_ids_3)
          if rq_is_robot_compliant:
              end_force_mode()
          end
      else:
          rq_move_norm_multi_grippers(rq_gripper_position, gripper_slave_ids_3)
      end
      # end: URCap Program Node
      $ 29 "SetPayloadNode: {PayloadReferenceComponent; InstallationPayloadComponent name=Payload_Empty; contributorInfo=com.ur.polyscope.payload.common.InstallationPayloadComponent$1@50a04d; mass=1.11 kg; centerOfGravity=(0.0, 0.0, 0.054); Ixx=0.001832, Iyy=0.001832, Izz=0.001832, Ixy=0.000000, Ixz=0.000000, Iyz=0.000000, transitionTime: 0.05 s}"
      set_target_payload(1.110000, [0.000000, 0.000000, 0.054000], [0.001832, 0.001832, 0.001832, 0.000000, 0.000000, 0.000000], 0.050000)
      $ 30 "Waypoint_7" "breakAfter"
      movel(Waypoint_7_p, a=1.2, v=0.25)
      # begin: URCap Program Node
      #   Source: Robotiq_Grippers, 3.19.1.111718, Robotiq Inc.
      #   Type: Gripper
      $ 31 "Gripper Close (1)"
      gripper_slave_ids_4 = [9]
      popupErrorGripperWord = "Gripper"
      popupErrorNoConnection1 = "must be connected to run this program."
      popupErrorNoConnection2 = "No connection"
      popupErrorNotActivated1 = "is not activated. Go to Installation tab > Gripper to activate it and run the program again."
      popupErrorNotActivated2 = "Not activated"
      rq_gripper_speed = 100.0
      rq_gripper_force = 100.0
      rq_gripper_position = 100.0
      rq_is_blocking = True
      rq_is_robot_compliant = False
      nb_slave_ids = get_list_length(gripper_slave_ids_4)
      rq_wait_for_gripper_reconnection()
      index = 0
      while (index < nb_slave_ids):
          if (not rq_is_gripper_connected(gripper_slave_ids_4[index])):
              write_error_popup(index, popupErrorGripperWord, popupErrorNoConnection1, popupErrorNoConnection2)
          end
          index = index + 1
      end
      index = 0
      while (index < nb_slave_ids):
          if (not rq_is_gripper_activated(gripper_slave_ids_4[index])):
              write_error_popup(index, popupErrorGripperWord, popupErrorNotActivated1, popupErrorNotActivated2)
          end
          index = index + 1
      end
      rq_set_speed_norm_multi_grippers(rq_gripper_speed, gripper_slave_ids_4)
      rq_set_force_norm_multi_grippers(rq_gripper_force, gripper_slave_ids_4)
      if (rq_is_blocking):
          if rq_is_robot_compliant:
              zero_ftsensor()
              sleep(0.02)
              # Maximum allowed deviation values for non-compliant axes are default values generated by UR in a Force node
              force_mode(tool_pose(), [1, 1, 0, 0, 0, 0], [0.0, 0.0, 0.0, 0.0, 0.0, 0.0], 2, [0.15, 0.15, 0.1, 0.3490658503988659, 0.3490658503988659, 0.3490658503988659])
          end
          rq_move_and_wait_norm_multi_grippers(rq_gripper_position, gripper_slave_ids_4)
          if rq_is_robot_compliant:
              end_force_mode()
          end
      else:
          rq_move_norm_multi_grippers(rq_gripper_position, gripper_slave_ids_4)
      end
      # end: URCap Program Node
      $ 32 "MoveL"
      $ 33 "Waypoint_11" "breakAfter"
      movel(Waypoint_11_p, a=1.2, v=0.25, r=0.01)
      $ 34 "Waypoint_12" "breakAfter"
      movel(Waypoint_12_p, a=1.2, v=0.25, r=0.01)
      $ 35 "Waypoint_13" "breakAfter"
      movel(Waypoint_13_p, a=1.2, v=0.25, r=0.01)
      $ 36 "Waypoint_14" "breakAfter"
      movel(Waypoint_14_p, a=1.2, v=0.25)
    else:
      $ 37 "Else" "noBreak"
      $ 38 "MoveL"
      $ 39 "Waypoint_8" "breakAfter"
      movel(Waypoint_8_p, a=1.2, v=0.25)
      # begin: URCap Program Node
      #   Source: Robotiq_Grippers, 3.19.1.111718, Robotiq Inc.
      #   Type: Gripper
      $ 40 "Gripper Open (1)"
      gripper_slave_ids_5 = [9]
      popupErrorGripperWord = "Gripper"
      popupErrorNoConnection1 = "must be connected to run this program."
      popupErrorNoConnection2 = "No connection"
      popupErrorNotActivated1 = "is not activated. Go to Installation tab > Gripper to activate it and run the program again."
      popupErrorNotActivated2 = "Not activated"
      rq_gripper_speed = 20.0
      rq_gripper_force = 100.0
      rq_gripper_position = 0.0
      rq_is_blocking = True
      rq_is_robot_compliant = False
      nb_slave_ids = get_list_length(gripper_slave_ids_5)
      rq_wait_for_gripper_reconnection()
      index = 0
      while (index < nb_slave_ids):
          if (not rq_is_gripper_connected(gripper_slave_ids_5[index])):
              write_error_popup(index, popupErrorGripperWord, popupErrorNoConnection1, popupErrorNoConnection2)
          end
          index = index + 1
      end
      index = 0
      while (index < nb_slave_ids):
          if (not rq_is_gripper_activated(gripper_slave_ids_5[index])):
              write_error_popup(index, popupErrorGripperWord, popupErrorNotActivated1, popupErrorNotActivated2)
          end
          index = index + 1
      end
      rq_set_speed_norm_multi_grippers(rq_gripper_speed, gripper_slave_ids_5)
      rq_set_force_norm_multi_grippers(rq_gripper_force, gripper_slave_ids_5)
      if (rq_is_blocking):
          if rq_is_robot_compliant:
              zero_ftsensor()
              sleep(0.02)
              # Maximum allowed deviation values for non-compliant axes are default values generated by UR in a Force node
              force_mode(tool_pose(), [1, 1, 0, 0, 0, 0], [0.0, 0.0, 0.0, 0.0, 0.0, 0.0], 2, [0.15, 0.15, 0.1, 0.3490658503988659, 0.3490658503988659, 0.3490658503988659])
          end
          rq_move_and_wait_norm_multi_grippers(rq_gripper_position, gripper_slave_ids_5)
          if rq_is_robot_compliant:
              end_force_mode()
          end
      else:
          rq_move_norm_multi_grippers(rq_gripper_position, gripper_slave_ids_5)
      end
      # end: URCap Program Node
      $ 41 "Waypoint_10" "breakAfter"
      movel(Waypoint_10_p, a=1.2, v=0.25)
      # begin: URCap Program Node
      #   Source: Robotiq_Grippers, 3.19.1.111718, Robotiq Inc.
      #   Type: Gripper
      $ 42 "Gripper Close (1)"
      gripper_slave_ids_6 = [9]
      popupErrorGripperWord = "Gripper"
      popupErrorNoConnection1 = "must be connected to run this program."
      popupErrorNoConnection2 = "No connection"
      popupErrorNotActivated1 = "is not activated. Go to Installation tab > Gripper to activate it and run the program again."
      popupErrorNotActivated2 = "Not activated"
      rq_gripper_speed = 20.0
      rq_gripper_force = 100.0
      rq_gripper_position = 100.0
      rq_is_blocking = True
      rq_is_robot_compliant = False
      nb_slave_ids = get_list_length(gripper_slave_ids_6)
      rq_wait_for_gripper_reconnection()
      index = 0
      while (index < nb_slave_ids):
          if (not rq_is_gripper_connected(gripper_slave_ids_6[index])):
              write_error_popup(index, popupErrorGripperWord, popupErrorNoConnection1, popupErrorNoConnection2)
          end
          index = index + 1
      end
      index = 0
      while (index < nb_slave_ids):
          if (not rq_is_gripper_activated(gripper_slave_ids_6[index])):
              write_error_popup(index, popupErrorGripperWord, popupErrorNotActivated1, popupErrorNotActivated2)
          end
          index = index + 1
      end
      rq_set_speed_norm_multi_grippers(rq_gripper_speed, gripper_slave_ids_6)
      rq_set_force_norm_multi_grippers(rq_gripper_force, gripper_slave_ids_6)
      if (rq_is_blocking):
          if rq_is_robot_compliant:
              zero_ftsensor()
              sleep(0.02)
              # Maximum allowed deviation values for non-compliant axes are default values generated by UR in a Force node
              force_mode(tool_pose(), [1, 1, 0, 0, 0, 0], [0.0, 0.0, 0.0, 0.0, 0.0, 0.0], 2, [0.15, 0.15, 0.1, 0.3490658503988659, 0.3490658503988659, 0.3490658503988659])
          end
          rq_move_and_wait_norm_multi_grippers(rq_gripper_position, gripper_slave_ids_6)
          if rq_is_robot_compliant:
              end_force_mode()
          end
      else:
          rq_move_norm_multi_grippers(rq_gripper_position, gripper_slave_ids_6)
      end
      # end: URCap Program Node
      $ 43 "SetPayloadNode: {PayloadReferenceComponent; InstallationPayloadComponent name=Payload_brick; contributorInfo=com.ur.polyscope.payload.common.InstallationPayloadComponent$1@50a04d; mass=1.18 kg; centerOfGravity=(0.003, -0.002, 0.05); Ixx=0.002028, Iyy=0.002028, Izz=0.002028, Ixy=0.000000, Ixz=0.000000, Iyz=0.000000, transitionTime: 0.05 s}"
      set_target_payload(1.180000, [0.003000, -0.002000, 0.050000], [0.002028, 0.002028, 0.002028, 0.000000, 0.000000, 0.000000], 0.050000)
      $ 44 "Waypoint_8" "breakAfter"
      movel(Waypoint_8_p, a=1.2, v=0.25)
      $ 45 "MoveJ"
      $ 46 "Waypoint_3" "breakAfter"
      movej(get_inverse_kin(Waypoint_3_p, qnear=Waypoint_3_q), a=1.3962634015954636, v=1.0471975511965976)
      $ 47 "Pallet_1"
      def Pallet_1_trans(pose):
      return p[pose[0], pose[1], pose[2], 0, 0, 0]
    end
    def Pallet_1_rot(pose):
    return p[0, 0, 0, pose[3], pose[4], pose[5]]
  end
  def Pallet_1_compute_pallet_waypoint(T_base_feature_taught, T_feature_referencePoint_taught, T_referencePoint_approach_taught, T_base_feature, T_base_referencePoint):
  local trans_referencePoint_approach_in_feature_taught = pose_sub(Pallet_1_trans(pose_trans(T_feature_referencePoint_taught, T_referencePoint_approach_taught)), Pallet_1_trans(T_feature_referencePoint_taught))
  local rot_referencePoint_approach_in_feature_taught = pose_trans(Pallet_1_rot(T_feature_referencePoint_taught), pose_trans(Pallet_1_rot(T_referencePoint_approach_taught), pose_inv(Pallet_1_rot(T_feature_referencePoint_taught))))
  T_feature_referencePoint = pose_trans(pose_inv(T_base_feature), T_base_referencePoint)
  rot_referencePoint_approach = pose_trans(pose_inv(Pallet_1_rot(T_feature_referencePoint)), pose_trans(rot_referencePoint_approach_in_feature_taught, Pallet_1_rot(T_feature_referencePoint)))
  T_feature_approach = pose_trans(trans_referencePoint_approach_in_feature_taught, pose_trans(T_feature_referencePoint, rot_referencePoint_approach))
  T_base_approach = pose_trans(T_base_feature, T_feature_approach)
  return T_base_approach
  end
  Pallet_1_tct = 6
  if (Pallet_1_cnt > 6 or Pallet_1_cnt < 1):
    Pallet_1_cnt = 1
  end
  $ 48 "Patterns" "noBreak"
  $ 49 "Grid_Pattern_1" "noBreak"
  $ 54 "Layers" "noBreak"
  if (Pallet_1_cnt < 7):
    Pallet_1_lno = 1
    Pallet_1_lct = Pallet_1_cnt
    global CornerItem_1=pose_trans(p[0.0,0.0,0.0,0.0,0.0,0.0], pose_trans(p[-.000000000000, -.000000000000, -.000000000000, .000000000000, .000000000000, .000000000000], p[.272815353413, -.001324543859, -.052174494010, .008705000024, -3.141549977485, .000049219086]))
    global CornerItem_2=pose_trans(p[0.0,0.0,0.0,0.0,0.0,0.0], pose_trans(p[-.000000000000, -.000000000000, -.000000000000, .000000000000, .000000000000, .000000000000], p[.390407517952, -.001340389777, -.053528308396, .008675688915, -3.141567407219, .000073299921]))
    global CornerItem_3=pose_trans(p[0.0,0.0,0.0,0.0,0.0,0.0], pose_trans(p[-.000000000000, -.000000000000, -.000000000000, .000000000000, .000000000000, .000000000000], p[.389560235333, .061974690253, -.053523155966, .008707500509, -3.141545639375, .000109832001]))
    global CornerItem_4=pose_trans(p[0.0,0.0,0.0,0.0,0.0,0.0], pose_trans(p[-.000000000000, -.000000000000, -.000000000000, .000000000000, .000000000000, .000000000000], p[.271914689512, .061973427774, -.054703295575, .008664201316, -3.141528694215, .000088930163]))
    Pallet_1_cnt_x = (Pallet_1_lct - 1) % 3
    Pallet_1_cnt_y = floor((Pallet_1_lct - 1) / 3)
    referencePoint = interpolate_pose(interpolate_pose(CornerItem_1, CornerItem_2, Pallet_1_cnt_x/2), interpolate_pose(CornerItem_4, CornerItem_3,Pallet_1_cnt_x/2), Pallet_1_cnt_y/1)
    if (Pallet_1_cnt_x < 1.5):
      if (Pallet_1_cnt_y < 1.0):
        qNearApproach = [0.5002027749876214, -1.5124365326845517, -2.2809078693381117, -0.9179548186049553, 1.5635657310591418, 2.060306787478332]
      else:
        qNearApproach = [0.7166069149837977, -1.5509234567045223, -2.2597515583062133, -0.9006658953386184, 1.5637841224774576, 2.276609897599947]
      end
    else:
      if (Pallet_1_cnt_y < 1.0):
        qNearApproach = [0.34201839567921954, -1.9967905483703507, -1.6839900016620497, -1.0305095476213308, 1.5646113157074673, 1.9031835794573944]
      else:
        qNearApproach = [0.49925589561185163, -2.01247229198513, -1.6595180034661094, -1.0393417042507336, 1.5646234750780454, 2.060486078260228]
      end
    end
    direction = p[0,0,1,0,0,0]
    referencePoint = pose_add (referencePoint,p[0.0*direction[0],0.0*direction[1],0.0*direction[2],0,0,0])
  end
  Approach_p = Pallet_1_compute_pallet_waypoint(p[0.0,0.0,0.0,0.0,0.0,0.0], pose_trans(pose_inv(p[0.0,0.0,0.0,0.0,0.0,0.0]), p[0.27281535341285135,-0.001324543859192466,-0.05217449401005958,0.00870500002447209,-3.141549977484781,4.9219085738482074E-5]), p[5.609244568272054E-7,-5.709052094625931E-7,-0.018268802801840053,0.0,0.0,0.0], p[0.0,0.0,0.0,0.0,0.0,0.0], referencePoint)
  Approach_p = pose_trans(p[0.27281535341285135,-0.001324543859192466,-0.05217449401005958,0.0087050000245021,-3.1415499774956595,4.921908569504902E-5], pose_trans(pose_inv(referencePoint), Approach_p))
  Approach_q = qNearApproach
  ToolActionPoint_p = Pallet_1_compute_pallet_waypoint(p[0.0,0.0,0.0,0.0,0.0,0.0], pose_trans(pose_inv(p[0.0,0.0,0.0,0.0,0.0,0.0]), p[0.27281535341285135,-0.001324543859192466,-0.05217449401005958,0.00870500002447209,-3.141549977484781,4.9219085738482074E-5]), p[0.0,4.3368086899420177E-19,-2.7755575615628914E-17,0.0,0.0,0.0], p[0.0,0.0,0.0,0.0,0.0,0.0], referencePoint)
  ToolActionPoint_p = pose_trans(p[0.27281535341285135,-0.001324543859192466,-0.05217449401005958,0.0087050000245021,-3.1415499774956595,4.921908569504902E-5], pose_trans(pose_inv(referencePoint), ToolActionPoint_p))
  Exit_1_p = Pallet_1_compute_pallet_waypoint(p[0.0,0.0,0.0,0.0,0.0,0.0], pose_trans(pose_inv(p[0.0,0.0,0.0,0.0,0.0,0.0]), p[0.27281535341285135,-0.001324543859192466,-0.05217449401005958,0.00870500002447209,-3.141549977484781,4.9219085738482074E-5]), p[2.997821961170377E-6,-3.0512485515218207E-6,-0.09764231465499425,0.0,0.0,0.0], p[0.0,0.0,0.0,0.0,0.0,0.0], referencePoint)
  Exit_1_p = pose_trans(p[0.27281535341285135,-0.001324543859192466,-0.05217449401005958,0.0087050000245021,-3.1415499774956595,4.921908569504902E-5], pose_trans(pose_inv(referencePoint), Exit_1_p))
  $ 55 "At Each Item" "noBreak"
  $ 56 "Generated Movements" "noBreak"
  $ 57 "MoveJ" "noBreak"
  $ 58 "Approach" "noBreak"
  movej(get_inverse_kin(pose_trans(referencePoint, pose_trans(p[.272805425444, .002834783509, -.052166206975, -.008705000024, 3.141549977488, -.000049219086], Approach_p)), qnear=Approach_q), a=1.3962634015954636, v=1.0471975511965976)
  $ 59 "MoveL" "noBreak"
  $ 60 "ToolActionPoint" "noBreak"
  movel(pose_trans(referencePoint, pose_trans(p[.272805425444, .002834783509, -.052166206975, -.008705000024, 3.141549977488, -.000049219086], ToolActionPoint_p)), a=1.2, v=0.25)
  $ 61 "Tool action" "noBreak"
  # begin: URCap Program Node
  #   Source: Robotiq_Grippers, 3.19.1.111718, Robotiq Inc.
  #   Type: Gripper
  $ 62 "Gripper Open (1)" "noBreak"
  gripper_slave_ids_7 = [9]
  popupErrorGripperWord = "Gripper"
  popupErrorNoConnection1 = "must be connected to run this program."
  popupErrorNoConnection2 = "No connection"
  popupErrorNotActivated1 = "is not activated. Go to Installation tab > Gripper to activate it and run the program again."
  popupErrorNotActivated2 = "Not activated"
  rq_gripper_speed = 20.0
  rq_gripper_force = 100.0
  rq_gripper_position = 0.0
  rq_is_blocking = True
  rq_is_robot_compliant = False
  nb_slave_ids = get_list_length(gripper_slave_ids_7)
  rq_wait_for_gripper_reconnection()
  index = 0
  while (index < nb_slave_ids):
      if (not rq_is_gripper_connected(gripper_slave_ids_7[index])):
          write_error_popup(index, popupErrorGripperWord, popupErrorNoConnection1, popupErrorNoConnection2)
      end
      index = index + 1
  end
  index = 0
  while (index < nb_slave_ids):
      if (not rq_is_gripper_activated(gripper_slave_ids_7[index])):
          write_error_popup(index, popupErrorGripperWord, popupErrorNotActivated1, popupErrorNotActivated2)
      end
      index = index + 1
  end
  rq_set_speed_norm_multi_grippers(rq_gripper_speed, gripper_slave_ids_7)
  rq_set_force_norm_multi_grippers(rq_gripper_force, gripper_slave_ids_7)
  if (rq_is_blocking):
      if rq_is_robot_compliant:
          zero_ftsensor()
          sleep(0.02)
          # Maximum allowed deviation values for non-compliant axes are default values generated by UR in a Force node
          force_mode(tool_pose(), [1, 1, 0, 0, 0, 0], [0.0, 0.0, 0.0, 0.0, 0.0, 0.0], 2, [0.15, 0.15, 0.1, 0.3490658503988659, 0.3490658503988659, 0.3490658503988659])
      end
      rq_move_and_wait_norm_multi_grippers(rq_gripper_position, gripper_slave_ids_7)
      if rq_is_robot_compliant:
          end_force_mode()
      end
  else:
      rq_move_norm_multi_grippers(rq_gripper_position, gripper_slave_ids_7)
  end
  # end: URCap Program Node
  $ 63 "SetPayloadNode: {PayloadReferenceComponent; InstallationPayloadComponent name=Payload_Empty; contributorInfo=com.ur.polyscope.payload.common.InstallationPayloadComponent$1@50a04d; mass=1.11 kg; centerOfGravity=(0.0, 0.0, 0.054); Ixx=0.001832, Iyy=0.001832, Izz=0.001832, Ixy=0.000000, Ixz=0.000000, Iyz=0.000000, transitionTime: 0.05 s}" "noBreak"
  set_target_payload(1.110000, [0.000000, 0.000000, 0.054000], [0.001832, 0.001832, 0.001832, 0.000000, 0.000000, 0.000000], 0.050000)
  $ 64 "MoveL" "noBreak"
  $ 65 "Exit_1" "noBreak"
  movel(pose_trans(referencePoint, pose_trans(p[.272805425444, .002834783509, -.052166206975, -.008705000024, 3.141549977488, -.000049219086], Exit_1_p)), a=1.2, v=0.25)
  Pallet_1_sep = False
  if (Pallet_1_cnt >= 6):
    Pallet_1_cnt = 1
  else:
    Pallet_1_cnt = Pallet_1_cnt + 1
  end
  end
  end
end
